{attribute 'qualified_only'}
{attribute 'strict'}
TYPE E_PState :
(
	Init, 
	SealIssue, 
	SealWait, 
	OpenValves, 
	Done, 
	Fault
);
END_TYPE

(* stored: Version 1.1.0.1, ProductVersion 3.1.4024.15
   DUT E_PState: Id {bfad5530-74f3-4942-8b59-c12de18475bb} *)
